# B&R Automation Studio project Bsp_Can_V001
Automation Studio 4.3.3.196

## Configuration Config1

CPU X20CP0482, AutomationRuntime D4.34, Build 4.1.2, Vc V4.34.1

### Task classes (Cpu.sw)
```
Cyclic#4:
  Program <- Program.prg
Libraries: CAN_Lib, runtime, Bsp_Can, Bsp_Alex
```

## Logical view

Binary libraries used (declarations not repeated): operator, runtime, astime, AsIecCon, CAN_Lib

### Package Logical/Libraries - 全局库

### Library Logical/Libraries/Bsp_Can (ANSIC)
Depends on: CAN_Lib

#### Constants.var - Exported constants
```iecst
VAR CONSTANT
	Mo : USINT := 1;
	Bg : USINT := 2;
	St : USINT := 3;
	Ac : USINT := 4;
	Dc : USINT := 5;
	Um : USINT := 6;
	Pa : USINT := 7;
	Pr : USINT := 8;
	Sp : USINT := 9;
	Jv : USINT := 10;
	Px : USINT := 11;
	Iq : USINT := 12;
	Ec : USINT := 13;
	Vx : USINT := 14;
END_VAR
```

#### Bsp_Can.fun - Exported functions and function blocks
```iecst
FUNCTION_BLOCK Can_Init (*TODO: 瞳늪警속팀쬠*) (*$GROUP=User,$CAT=User,$GROUPICON=User.png,$CATICON=User.png*)
	VAR_INPUT
		wDevice : UDINT;
		wModule_Id : ARRAY[0..2] OF USINT;
	END_VAR
	VAR_OUTPUT
		rUs_Ident : UDINT;
		rQ_Ident : ARRAY[0..2] OF UDINT;
		rErr_Code : UINT;
	END_VAR
END_FUNCTION_BLOCK

FUNCTION_BLOCK Can_Write (*TODO: 瞳늪警속팀쬠*) (*$GROUP=User,$CAT=User,$GROUPICON=User.png,$CATICON=User.png*)
	VAR_INPUT
		wModule_Id : USINT;
		wUs_Ident : UDINT;
		wData_Adr : UDINT;
		wLen : USINT;
	END_VAR
	VAR_OUTPUT
		rErr_Code : UINT;
	END_VAR
END_FUNCTION_BLOCK

FUNCTION_BLOCK Set_Motor (*TODO: 瞳늪警속팀쬠*) (*$GROUP=User,$CAT=User,$GROUPICON=User.png,$CATICON=User.png*)
	VAR_INPUT
		wCmd : USINT;
		wModule_Id : USINT;
		wUs_Ident : UDINT;
		wValue : UDINT;
	END_VAR
	VAR_OUTPUT
		rErr_Code : UINT;
	END_VAR
END_FUNCTION_BLOCK

FUNCTION_BLOCK Get_Motor (*TODO: 瞳늪警속팀쬠*) (*$GROUP=User,$CAT=User,$GROUPICON=User.png,$CATICON=User.png*)
	VAR_INPUT
		wQ_Ident : UDINT;
		wUs_Ident : UDINT;
		wModule_Id : USINT;
	END_VAR
	VAR_OUTPUT
		rErr_Code : UINT;
		rActSpeed : DINT;
		rActCurrent : INT;
		rDrvMode : USINT;
		rEncCount : DINT;
	END_VAR
END_FUNCTION_BLOCK

FUNCTION Set_Arry : BOOL
	VAR_INPUT
		data_adr : REFERENCE TO USINT;
		_a : USINT;
		_b_ : USINT;
		_c : USINT;
		_d : USINT;
		_e : USINT;
		_f : USINT;
		_g : USINT;
		_h : USINT;
	END_VAR
END_FUNCTION
```

#### Can_Init.c
```c
#include <bur/plctypes.h>
#ifdef __cplusplus
	extern "C"
	{
#endif
	#include "Bsp_Can.h"
#ifdef __cplusplus
	};
#endif
/* TODO: 瞳늪警속팀쬠 */
void Can_Init(struct Can_Init* inst)
{
	CANopen_typ CANopen_0;
	CANqueue_typ CANqueue_0;
	CANqueue_typ CANqueue_1;
	CANqueue_typ CANqueue_2;
	CANquwr_typ CANquwr_0;

	USINT _data[] = {0x01, 0x00};

	CANopen_0.enable = 1;
	CANopen_0.baud_rate = 50;
	CANopen_0.cob_anz = 5;
	CANopen_0.device = (UDINT)inst->wDevice;
	CANopen_0.info = 0;
	CANopen(&CANopen_0);
	inst->rErr_Code = CANopen_0.status;
	inst->rUs_Ident = CANopen_0.us_ident;

	CANqueue_0.enable = 1;
	CANqueue_0.us_ident = CANopen_0.us_ident;
	CANqueue_0.can_id = 0x280 + inst->wModule_Id[0];;
	CANqueue_0.size = 20;
	CANqueue(&CANqueue_0);
	inst->rErr_Code = CANqueue_0.status;
	inst->rQ_Ident[0] = CANqueue_0.q_ident;

	CANqueue_1.enable = 1;
	CANqueue_1.us_ident = CANopen_0.us_ident;
	CANqueue_1.can_id = 0x280 + inst->wModule_Id[1];
	CANqueue_1.size = 20;
	CANqueue(&CANqueue_0);
	inst->rErr_Code = CANqueue_1.status;
	inst->rQ_Ident[1] = CANqueue_1.q_ident;

	CANqueue_2.enable = 1;
	CANqueue_2.us_ident = CANopen_0.us_ident;
	CANqueue_2.can_id = 0x280 + inst->wModule_Id[2];
	CANqueue_2.size = 20;
	CANqueue(&CANqueue_0);
	inst->rErr_Code = CANqueue_2.status;
	inst->rQ_Ident[2] = CANqueue_2.q_ident;

	CANquwr_0.enable = 1;
	CANquwr_0.us_ident = CANopen_0.us_ident;;
	CANquwr_0.can_id = 0x000;
	CANquwr_0.data_adr = (UDINT)_data;
	CANquwr_0.data_lng = 2;
	CANquwr(&CANquwr_0);
	inst->rErr_Code = CANquwr_0.status;
}
```

#### Can_Write.c
```c
#include <bur/plctypes.h>
#ifdef __cplusplus
	extern "C"
	{
#endif
	#include "Bsp_Can.h"
#ifdef __cplusplus
	};
#endif
/* TODO: 瞳늪警속팀쬠 */
void Can_Write(struct Can_Write* inst)
{
	CANquwr_typ CANquwr_0;

	CANquwr_0.enable = 1;
	CANquwr_0.us_ident = inst->wUs_Ident;
	CANquwr_0.can_id = 0x300 + inst->wModule_Id;
	CANquwr_0.data_adr = inst->wData_Adr;
	CANquwr_0.data_lng = inst->wLen;
	CANquwr(&CANquwr_0);

	inst->rErr_Code = CANquwr_0.status;
}
```

#### Set_Motor.c
```c
#include <bur/plctypes.h>
#ifdef __cplusplus
	extern "C"
	{
#endif
	#include "Bsp_Can.h"
#ifdef __cplusplus
	};
#endif
/* TODO: 瞳늪警속팀쬠 */
void Set_Motor(struct Set_Motor* inst)
{
	USINT _data[8];
	struct Can_Write CanWrite_0;
	switch (inst->wCmd)
	{
		case Mo:	Set_Arry(_data, 0x4D, 0x4F, 0x00, 0x00, (USINT)inst->wValue, 0x00, 0x00, 0x00);
			CanWrite_0.wLen = 8;
			break;

		case Bg:	Set_Arry(_data, 0x42, 0x47, 0x00, 0x00, 0x00, 0x00, 0x00, 0x00);
			CanWrite_0.wLen = 4;
			break;

		case St:	Set_Arry(_data, 0x53, 0x54, 0x00, 0x00, 0x00, 0x00, 0x00, 0x00);
			CanWrite_0.wLen = 4;
			break;

		case Ac:	Set_Arry(_data, 0x41, 0x43, 0x00, 0x00, (USINT)(inst->wValue % 256 % 256), (USINT)(inst->wValue % 256 / 256), (USINT)(inst->wValue / 256 / 256), 0x00);
			CanWrite_0.wLen = 8;
			break;

		case Dc:	Set_Arry(_data, 0x44, 0x43, 0x00, 0x00, (USINT)(inst->wValue % 256 % 256), (USINT)(inst->wValue % 256 / 256), (USINT)(inst->wValue / 256 / 256), 0x00);
			CanWrite_0.wLen = 8;
			break;

		case Um:	Set_Arry(_data, 0x55, 0x4D, 0x00, 0x00, inst->wValue, 0x00, 0x00, 0x00);
			CanWrite_0.wLen = 8;
			break;

		case Pa:	Set_Arry(_data, 0x50, 0x41, 0x00, 0x00, (USINT)(inst->wValue % 256), (USINT)(inst->wValue / 256), 0x00, 0x00);
			CanWrite_0.wLen = 8;
			break;

		case Pr:	Set_Arry(_data, 0x50, 0x52, 0x00, 0x00, (USINT)(inst->wValue % 256), (USINT)(inst->wValue / 256), 0x00, 0x00);
			CanWrite_0.wLen = 8;
			break;

		case Sp:	Set_Arry(_data, 0x53, 0x50, 0x00, 0x00, (USINT)(inst->wValue % 256), (USINT)(inst->wValue / 256), 0x00, 0x00);
			CanWrite_0.wLen = 8;
			break;

		case Jv:	Set_Arry(_data, 0x4A, 0x56, 0x00, 0x00, (USINT)(inst->wValue % 256), (USINT)(inst->wValue / 256), 0x00, 0x00);
			CanWrite_0.wLen = 8;
			break;

		case Px:	Set_Arry(_data, 0x50, 0x58, 0x00, 0x00, (USINT)(inst->wValue % 256), (USINT)(inst->wValue / 256), 0x00, 0x00);
			CanWrite_0.wLen = 8;
			break;

		default:	break;

	}
	CanWrite_0.wUs_Ident = inst->wUs_Ident;
	CanWrite_0.wModule_Id = inst->wModule_Id;
	CanWrite_0.wData_Adr = (UDINT)_data;

	Can_Write(&CanWrite_0);

	inst->rErr_Code = CanWrite_0.rErr_Code;

}

BOOL Set_Arry(USINT *data_adr, USINT _a, USINT _b, USINT _c, USINT _d, USINT _e, USINT _f, USINT _g, USINT _h)
{
	*(data_adr + 0) = _a;
	*(data_adr + 1) = _b;
	*(data_adr + 2) = _c;
	*(data_adr + 3) = _d;
	*(data_adr + 4) = _e;
	*(data_adr + 5) = _f;
	*(data_adr + 6) = _g;
	*(data_adr + 7) = _h;
	return 0;
}
```

#### Get_Motor.c
```c
#include <bur/plctypes.h>
#ifdef __cplusplus
	extern "C"
	{
#endif
	#include "Bsp_Can.h"
#ifdef __cplusplus
	};
#endif
/* TODO: 瞳늪警속팀쬠 */
void Get_Motor(struct Get_Motor* inst)
{
	CANrd_typ CANrd_0;
	struct Can_Write Can_Write_0;
	USINT _temp[4];
	USINT _cmd[4];
	USINT i;

	CANrd_0.enable = 1;
	CANrd_0.q_ident = inst->wQ_Ident;
	CANrd_0.data_adr = (UDINT)_temp;

	Can_Write_0.wUs_Ident = inst->wUs_Ident;
	Can_Write_0.wModule_Id = inst->wModule_Id;

	//꿴璂JV
	Set_Arry(_cmd, 0x4A, 0x56, 0x00, 0x00, 0x00, 0x00, 0x00, 0x00);
	Can_Write_0.wData_Adr = (UDINT)_cmd;
	Can_Write_0.wLen = 4;
	Can_Write(&Can_Write_0);
	//꿴璂IQ
	Set_Arry(_cmd, 0x49, 0x51, 0x00, 0x00, 0x00, 0x00, 0x00, 0x00);
	Can_Write_0.wData_Adr = (UDINT)_cmd;
	Can_Write_0.wLen = 4;
	Can_Write(&Can_Write_0);
	//꿴璂UM
	Set_Arry(_cmd, 0x4A, 0x56, 0x00, 0x00, 0x00, 0x00, 0x00, 0x00);
	Can_Write_0.wData_Adr = (UDINT)_cmd;
	Can_Write_0.wLen = 4;
	Can_Write(&Can_Write_0);
	//꿴璂PX
	Set_Arry(_cmd, 0x4A, 0x56, 0x00, 0x00, 0x00, 0x00, 0x00, 0x00);
	Can_Write_0.wData_Adr = (UDINT)_cmd;
	Can_Write_0.wLen = 4;
	Can_Write(&Can_Write_0);

	for(i=0; i<4; i++)
	{
		CANrd(&CANrd_0);
		inst->rErr_Code = CANrd_0.status;

		if((_temp[0]==0x4A) && (_temp[1]==0x56))//JV
			inst->rActSpeed = _temp[5] * 256 + _temp[4];
		else if((_temp[0]==0x49) && (_temp[1]==0x51))//IQ
			inst->rActCurrent = _temp[5] * 256 + _temp[4];
		else if((_temp[0]==0x55) && (_temp[1]==0x4D))//UM
			inst->rDrvMode = _temp[4];
		else if((_temp[0]==0x50) && (_temp[1]==0x58))//PX
			inst->rEncCount = _temp[5] * 256 + _temp[4];

	}
}
```

### Library Logical/Libraries/Bsp_Alex (ANSIC)
Depends on: Bsp_Can

#### Types.typ - Exported data types
```iecst
TYPE
	ProPosMode_type : 	STRUCT
		wRel : BOOL;
		wAbs : BOOL;
		wTargetPos : DINT;
		wProVloc : UDINT;
	END_STRUCT;
	ProVelMode_type : 	STRUCT
		wSetSpd : DINT;
	END_STRUCT;
	ElmoMotor : 	STRUCT
		wCINH : BOOL;
		wQSP : BOOL;
		wProAclera : UDINT;
		wProDeclera : UDINT;
		wDrvMode : SINT;
		wOpMode1 : ProPosMode_type;
		wOpMode3 : ProVelMode_type;
		rActSpeed : DINT;
		rActCurrent : INT;
		rDrvMode : USINT;
		rEncCount : DINT;
		rErrCode : UINT;
		rCommOK : BOOL;
	END_STRUCT;
END_TYPE
```

#### Bsp_Alex.fun - Exported functions and function blocks
```iecst
FUNCTION_BLOCK Update_ElmoMotor
	VAR_INPUT
		ElmoMotor_0 : {REDUND_UNREPLICABLE} ElmoMotor;
		wUs_Ident : UDINT;
		wQ_Ident : UDINT;
		wModule_Id : USINT;
	END_VAR
	VAR_OUTPUT
		rErr_Code : UINT;
	END_VAR
END_FUNCTION_BLOCK
```

#### Update_ElmoMotor.c
```c
#include <bur/plctypes.h>
#ifdef __cplusplus
	extern "C"
	{
#endif
	#include "Bsp_Alex.h"
#ifdef __cplusplus
	};
#endif
/* TODO: 瞳늪警속팀쬠 */
void Update_ElmoMotor(struct Update_ElmoMotor* inst)
{
	struct Set_Motor Set_Motor_0;
	struct Get_Motor Get_Motor_0;

	Set_Motor_0.wUs_Ident = inst->wUs_Ident;
	Set_Motor_0.wModule_Id = inst->wModule_Id;

	//MO
	Set_Motor_0.wCmd = Mo;
	Set_Motor_0.wValue = inst->ElmoMotor_0.wCINH;
	Set_Motor(&Set_Motor_0);
	inst->rErr_Code = Set_Motor_0.rErr_Code;

	//ST
	if(inst->ElmoMotor_0.wQSP == 1)
	{
		Set_Motor_0.wCmd = St;
		Set_Motor(&Set_Motor_0);
		inst->rErr_Code = Set_Motor_0.rErr_Code;
	}

	//AC
	Set_Motor_0.wCmd = Pa;
	Set_Motor_0.wValue = inst->ElmoMotor_0.wProAclera;
	Set_Motor(&Set_Motor_0);
	inst->rErr_Code = Set_Motor_0.rErr_Code;

	//DC
	Set_Motor_0.wCmd = Pa;
	Set_Motor_0.wValue = inst->ElmoMotor_0.wProDeclera;
	Set_Motor(&Set_Motor_0);
	inst->rErr_Code = Set_Motor_0.rErr_Code;

	//UM
	Set_Motor_0.wCmd = Um;
	Set_Motor_0.wValue = inst->ElmoMotor_0.wDrvMode;
	Set_Motor(&Set_Motor_0);
	inst->rErr_Code = Set_Motor_0.rErr_Code;

	//PR
	if(inst->ElmoMotor_0.wOpMode1.wRel == 1)
	{
		Set_Motor_0.wCmd = Pr;
		Set_Motor_0.wValue = inst->ElmoMotor_0.wOpMode1.wTargetPos;
		Set_Motor(&Set_Motor_0);
		inst->rErr_Code = Set_Motor_0.rErr_Code;
	}
	//PA
	else if(inst->ElmoMotor_0.wOpMode1.wAbs == 1)
	{
		Set_Motor_0.wCmd = Pa;
		Set_Motor_0.wValue = inst->ElmoMotor_0.wOpMode1.wTargetPos;
		Set_Motor(&Set_Motor_0);
		inst->rErr_Code = Set_Motor_0.rErr_Code;
	}
	//SP
	Set_Motor_0.wCmd = Sp;
	Set_Motor_0.wValue = inst->ElmoMotor_0.wOpMode1.wProVloc;
	Set_Motor(&Set_Motor_0);
	inst->rErr_Code = Set_Motor_0.rErr_Code;

	//JV
	Set_Motor_0.wCmd = Jv;
	Set_Motor_0.wValue = inst->ElmoMotor_0.wOpMode3.wSetSpd;
	Set_Motor(&Set_Motor_0);
	inst->rErr_Code = Set_Motor_0.rErr_Code;

	Get_Motor_0.wUs_Ident = inst->wUs_Ident;
	Get_Motor_0.wQ_Ident = inst->wQ_Ident;
	Get_Motor_0.wModule_Id = inst->wModule_Id;
	Get_Motor(&Get_Motor_0);

	inst->ElmoMotor_0.rActSpeed = Get_Motor_0.rActSpeed;
	inst->ElmoMotor_0.rActCurrent = Get_Motor_0.rActCurrent;
	inst->ElmoMotor_0.rDrvMode = Get_Motor_0.rDrvMode;
	inst->ElmoMotor_0.rEncCount = Get_Motor_0.rEncCount;
}
```

### Program Logical/Program (ANSIC)

#### Cyclic.c - Cyclic code
```c
#include <bur/plctypes.h>

#ifdef _DEFAULT_INCLUDES
	#include <AsDefault.h>
#endif

void _CYCLIC ProgramCyclic(void)
{
	if(Begin_Flag == 1)
	{
		Can_Init_0.wDevice = (UDINT)"IF7";
		Can_Init_0.wModule_Id[0] = 0x0B;
		Can_Init(&Can_Init_0);

		ElmoMotor_0.wCINH = 1;
		ElmoMotor_0.wDrvMode = 5;

		Update_ElmoMotor_0.ElmoMotor_0 = ElmoMotor_0;
		Update_ElmoMotor_0.wUs_Ident = Can_Init_0.rUs_Ident;
		Update_ElmoMotor_0.wQ_Ident = Can_Init_0.rQ_Ident[0];
		Update_ElmoMotor_0.wModule_Id = 0x0B;

		Begin_Flag = 0;
	}

	Update_ElmoMotor(&Update_ElmoMotor_0);
}
```

#### Variables.var - Local variables
```iecst
VAR
	Can_Init_0 : Can_Init;
	ElmoMotor_0 : ElmoMotor;
	Update_ElmoMotor_0 : Update_ElmoMotor;
	Begin_Flag : BOOL := TRUE;
END_VAR
```

Listed in the project but not available here: Logical/Global.typ, Logical/Global.var, Logical/Libraries/Bsp_Can/Types.typ, Logical/Libraries/Bsp_Alex/Constants.var, Logical/Program/Init.c, Logical/Program/Exit.c, Logical/Program/Types.typ
